FUNCTION_BLOCK RGBW
VAR_INPUT
END_VAR
VAR_OUTPUT
END_VAR
VAR
	Red		AT%Q*	:	INT;
	Green	AT%Q*	:	INT;
	Blue	AT%Q*	:	INT;
	White	AT%Q*	:	INT;
		
	Run		:	BOOL;
	
	ton		:	TON;
	Delay	:	TIME := T#0.5S;
	
	Countdown	:	INT		:= 5;
	On			:	BOOL	:= FALSE;;
END_VAR

IF Run THEN
	ton.IN := NOT ton.Q;
	ton.PT := Delay;
	
	IF ton.Q AND Countdown > 0 THEN //flashes 5 amber lights at < 1 second delay
		IF NOT On THEN
			Red := 32767;
			Green := 15000;
			Countdown := Countdown - 1;
			On := TRUE;
		ELSIF On THEN
			Red := 0;
			Green := 0;
			On := FALSE;
		END_IF
	ELSIF ton.Q AND Countdown = 0 THEN //go green lights 2 second delay
		Green := 32767;
		Red := 0;
		Countdown := -1;
	ELSIF ton.Q AND Countdown < 0 THEN //turns off countdown and resets counter after 2 seconds of green
		Run := FALSE;
	END_IF
	
	IF Countdown = 0 THEN
		Delay := T#2S;
	END_IF
	
	ton();
ELSIF NOT Run THEN
	Red := 0;
	Green := 0;
	Blue := 0;
	White := 0;
	Countdown := 5;
	Delay := T#0.5S;
END_IF

END_FUNCTION_BLOCK

(* stored: Version 1.1.0.1, ProductVersion 3.1.4024.12
   POU RGBW: Id {ae082d2a-8caf-460c-9c60-3ce2027f41cd}, SpecialFunc None *)
